FUNCTION TryConvert_USINT_TO_DT : BOOL
VAR_INPUT
	in : USINT;
	out : REFERENCE TO DT;
END_VAR

out := USINT_TO_DT(in);
TryConvert_USINT_TO_DT := TRUE;

END_FUNCTION

(* stored: Version 1.1.0.1, ProductVersion 3.1.4024.12
   POU TryConvert_USINT_TO_DT: Id {8f56a281-9ea2-4953-bc32-296f0b0ba987}, SpecialFunc None *)
